FUNCTION_BLOCK FB_AnalogInputThermocouple EXTENDS FB_DigitalDevice// use for El 3314
VAR
	iRawValue	AT%I*: INT;
	lrSclale : LREAL := 0.1;
	lrValue	: LREAL;
	bError		AT%I* : BOOL;
	
END_VAR

lrValue := INT_TO_LREAL(iRawValue)*lrSclale;

PROPERTY Error :  bool
GET
Error := bError;
END_GET
END_PROPERTY

PROPERTY Scale : lreal // Value = rawValue form terminal * scale
GET
Scale := lrSclale;
END_GET
SET
lrSclale := Scale;
END_SET
END_PROPERTY

{attribute 'monitoring' := 'variable'}
PROPERTY Value : REFERENCE TO  lreal
GET
Value ref= lrValue;
END_GET
END_PROPERTY

END_FUNCTION_BLOCK

(* stored: Version 1.1.0.1, ProductVersion 3.1.4024.12
   POU FB_AnalogInputThermocouple: Id {b85ab3fe-f3eb-4327-9ef8-a140d597c9c1}, SpecialFunc None
   Folder Properties: Id {5cf42921-bbce-4702-97a5-1a99b4a0783b}
   Property Error: Id {ab2e1c44-95b0-4ebc-94e8-615ac7269816}
   Get Get: Id {bda8db2e-1e74-4319-afff-ff0f41d9c0b7}
   Property Scale: Id {2e0c16de-5464-4cc7-a842-5343f66e8a06}
   Get Get: Id {3e56ef36-6590-4693-a2e1-2ede761b621d}
   Set Set: Id {eeadc2bd-2686-47d0-8a57-718c35b02cd1}
   Property Value: Id {56861794-75ed-4812-9d3b-6dd02f1ebe67}
   Get Get: Id {2b4a1990-be09-4658-8576-10da6ebbc964} *)
